ABB RobotStudio station: CeldaRobotica_PurpleWood.rsstnx

Station CeldaRobotica_PurpleWood (saved by RobotStudio 22.3.10190.2)
Controller Controlador1, task T_ROB1: task frame (RAPID world) sits at (-200, -100, 255) mm in the station
Controller Controlador1
  mechanical unit ROB_1: IRB1600_6_145__02, 6 joints, base frame (0, 0, 0) mm
Layout (positions relative to the parent item):
  - SC_Conveyor [smart component]
      signals: DI Crear_Gato, DI Crear_Estante, DI Crear_Mesa, DO DO_HIGH, DO DO_MID, DO DO_LOW, DO DO_GIRO
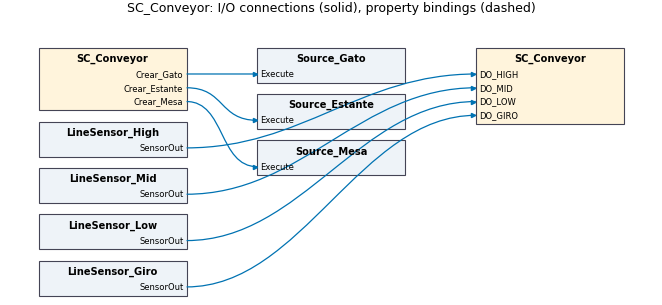
      connections:
        SC_Conveyor.Crear_Gato -> Source_Gato.Execute
        SC_Conveyor.Crear_Estante -> Source_Estante.Execute
        SC_Conveyor.Crear_Mesa -> Source_Mesa.Execute
        LineSensor_High.SensorOut -> SC_Conveyor.DO_HIGH
        LineSensor_Mid.SensorOut -> SC_Conveyor.DO_MID
        LineSensor_Low.SensorOut -> SC_Conveyor.DO_LOW
        LineSensor_Giro.SensorOut -> SC_Conveyor.DO_GIRO
    - EstanteColgado [graphiccomponentgroup] at (1130, -1000, 1506.1) mm, rotated rx 0 ry 0 rz 90 deg
      - RepisaLego:1 [graphiccomponentgroup] at (-95.35, -24.33, -484.95) mm, rotated rx 90 ry 86.54 rz -90 deg
        - RLV1 Fondo:1 [part] at (-151.16, -62.59, -80.25) mm, rotated rx 0 ry 90 rz 0 deg, size 66.4 x 11.1 x 483.7 mm
        - RLV1 Frente:1 [part] at (-151.16, -22.59, -49.25) mm, rotated rx 90 ry 0 rz 90 deg, size 83.3 x 30 x 483.3 mm
        - RLV1 Lateral:1 [part] at (-382.16, -18.58, -80.25) mm, rotated rx 180 ry 0 rz 180 deg, size 10.1 x 72.1 x 63.1 mm
        - RLV1 Trasera:1 [part] at (-151.16, -22.59, -111.25) mm, rotated rx -90 ry 0 rz 90 deg, size 91.4 x 15.2 x 487.6 mm
        - RLV1 Lateral:2 [part] at (88.84, -18.58, -80.25) mm, rotated rx 180 ry 0 rz 180 deg, size 10.1 x 72.1 x 63.1 mm
      - Gancho:1 [part] at (0, 0, -143.1) mm, size 142.1 x 142.1 x 242.6 mm
    - MesaColgada [graphiccomponentgroup] at (1130, -1000, 1506.1) mm, rotated rx 0 ry 0 rz 90 deg
      - AssemblyMesa2:1 [graphiccomponentgroup] at (0.6, -56.61, -255.15) mm, rotated rx -90 ry 79.48 rz -90 deg
        - MV1 Pata:1 [part] at (317.81, 42.68, -57.5) mm, size 36.5 x 51.1 x 116.8 mm
        - MV1 Tabla:1 [part] at (61.67, 51.7, 0) mm, rotated rx -90 ry 0 rz 0 deg, size 503.6 x 139.7 x 18.4 mm
        - MV1 Pata_MIR:1 [part] at (-194.43, 42.68, -57.5) mm, rotated rx 180 ry 0 rz 180 deg, size 36.5 x 51.1 x 116.8 mm
      - Gancho:1 [part] at (0, 0, -143.1) mm, size 142.1 x 142.1 x 242.6 mm
      - Source_Gato [smart component, from Components\Source.rslib] at (1000, 1130, -1506.1) mm, rotated rx 0 ry 0 rz -90 deg
          properties: Source=(none); Copy=(none); Parent=(none); Position=[0 0 0]; Orientation=[0 0 0]; Transient=false; PhysicsBehavior=-1
    - CasaGatoColgada_2 [graphiccomponentgroup] at (1130, -1000, 1506.1) mm, rotated rx 0 ry 0 rz 90 deg
      - Gancho:1 [part] at (0, 0, -143.1) mm, size 142.1 x 142.1 x 242.6 mm
      - CGV1 Pieza Base:1 [part] at (-126.11, -5.04, -68.58) mm, rotated rx -1.14 ry 0 rz 0 deg, size 304.2 x 16.3 x 706.2 mm
    - Source_Mesa [smart component, from Components\Source.rslib]
        properties: Source=MesaColgada; Copy=(none); Parent=(none); Position=[1.13 -2.9 1.5061]; Orientation=[0 0 1.5707963267949]; Transient=true; PhysicsBehavior=3
    - Source_Estante [smart component, from Components\Source.rslib]
        properties: Source=EstanteColgado; Copy=(none); Parent=(none); Position=[1.13 -2.9 1.5061]; Orientation=[0 0 1.5707963267949]; Transient=true; PhysicsBehavior=3
    - PhysicsControl [smart component, from Components\PhysicsControl.rslib]
        properties: Object=ConveyorAux; Behavior=1; SurfaceVelocity=0.05
    - LineSensor_Low [smart component, from Components\LineSensor.rslib]
        properties: Start=[1.2 -0.8 0.8]; End=[1.1 -0.8 0.8]; Radius=0; SensedPart=(none); SensedPoint=[0 0 0]
      - _sensorPart_ [part], size 100 x 0 x 0 mm
    - LineSensor_Mid [smart component, from Components\LineSensor.rslib]
        properties: Start=[1.15 -0.8 0.95]; End=[1.1 -0.8 0.95]; Radius=0; SensedPart=(none); SensedPoint=[0 0 0]
      - _sensorPart_ [part], size 50 x 0 x 0 mm
    - LineSensor_High [smart component, from Components\LineSensor.rslib]
        properties: Start=[1.3 -0.8 0.95]; End=[1.2 -0.8 0.95]; Radius=0; SensedPart=(none); SensedPoint=[0 0 0]
      - _sensorPart_ [part], size 100 x 0 x 0 mm
    - Source_Gato [smart component, from Components\Source.rslib]
        properties: Source=CasaGatoColgada_2; Copy=(none); Parent=(none); Position=[1.13 -2.9 1.5061]; Orientation=[0 0 1.5707963267949]; Transient=true; PhysicsBehavior=3
    - PhysicsControl_2 [smart component, from Components\PhysicsControl.rslib]
        properties: Object=ConveyorAux2; Behavior=1; SurfaceVelocity=0.05
    - ConveyorAux [part], size 30 x 6000 x 30 mm
    - ConveyorAux2 [part], size 30 x 6000 x 30 mm
    - LineSensor_Giro [smart component, from Components\LineSensor.rslib]
        properties: Start=[1.2 0 1.55]; End=[1.1 0 1.55]; Radius=0; SensedPart=(none); SensedPoint=[0 0 0]
      - _sensorPart_ [part], size 100 x 0 x 0 mm
  - Robotpedestal1400_H240 [part, from Equipment\Robot Pedestal 1400 H240.rslib] at (-330, -100, 0) mm
  - IRB1600_6_145__02 [mechanism, from Robots\IRB1600_6_145_G_02.rslib] at (-200, -100, 255) mm; joint values [0.1049, 0.2988, -0.3505, -0.1652, 0.584, 0.1908] (rad or m)
  - Conveyor [part], size 71 x 6000 x 68 mm
  - MyNewTool [mechanism] at (806.29, 0, 1409) mm, rotated rx -180 ry 60 rz -180 deg
      TCP MyNewTool at (0, 0, 200) mm
      links: Pieza_1
  - Fence_2500 [graphiccomponentgroup, from Equipment\Fence_2500.rslib] at (800, 1500, 0) mm, rotated rx 0 ry 0 rz 90 deg
    - Body 1 [part, from Equipment\Fence_2500.rslib]
    - Body 2 [part, from Equipment\Fence_2500.rslib]
  - Fence_2500_2 [graphiccomponentgroup, from Equipment\Fence_2500.rslib] at (1500, -1000, 0) mm
    - Body 1 [part, from Equipment\Fence_2500.rslib]
    - Body 2 [part, from Equipment\Fence_2500.rslib]
  - Fence_2500_3 [graphiccomponentgroup, from Equipment\Fence_2500.rslib] at (-1800, -1000, 0) mm
    - Body 1 [part, from Equipment\Fence_2500.rslib]
    - Body 2 [part, from Equipment\Fence_2500.rslib]
  - Gate [graphiccomponentgroup, from Equipment\Fence_Gate.rslib] at (-300, -1800, 0) mm, rotated rx 0 ry 0 rz 90 deg
    - Body 1 [part, from Equipment\Fence_Gate.rslib]
    - Body 2 [part, from Equipment\Fence_Gate.rslib]
    - Body 3 [part, from Equipment\Fence_Gate.rslib]
  - Fence_740 [graphiccomponentgroup, from Equipment\Fence_740.rslib] at (-1800, -1750, 0) mm
    - Body 1 [part, from Equipment\Fence_740.rslib]
    - Body 2 [part, from Equipment\Fence_740.rslib]
  - Fence_740_2 [graphiccomponentgroup, from Equipment\Fence_740.rslib] at (500, -1800, 0) mm, rotated rx 0 ry 0 rz 90 deg
    - Body 1 [part, from Equipment\Fence_740.rslib]
    - Body 2 [part, from Equipment\Fence_740.rslib]
  - Fence_740_3 [graphiccomponentgroup, from Equipment\Fence_740.rslib] at (1500, -1800, 0) mm
    - Body 1 [part, from Equipment\Fence_740.rslib]
    - Body 2 [part, from Equipment\Fence_740.rslib]
  - IRC5_Singel-Cabinet [part, from Equipment\IRC5_Singel-Cabinet.rslib] at (-2350, -1400, 100) mm, rotated rx 90 ry 0 rz -90 deg
Attachment: MyNewTool is attached to IRB1600_6_145__02 / Link6
Station signals: DO Estado_Pistola
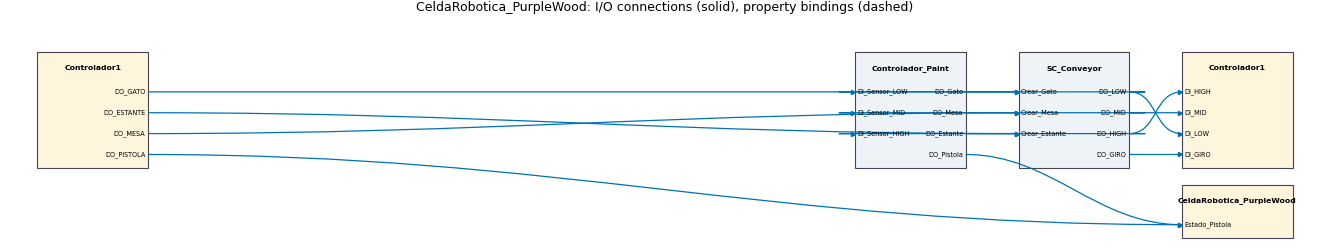
Station logic (signal -> signal, property => property):
  SC_Conveyor.DO_LOW -> Controlador_Paint.DI_Sensor_LOW
  SC_Conveyor.DO_MID -> Controlador_Paint.DI_Sensor_MID
  SC_Conveyor.DO_HIGH -> Controlador_Paint.DI_Sensor_HIGH
  Controlador_Paint.DO_Gato -> SC_Conveyor.Crear_Gato
  Controlador_Paint.DO_Mesa -> SC_Conveyor.Crear_Mesa
  Controlador_Paint.DO_Estante -> SC_Conveyor.Crear_Estante
  Controlador_Paint.DO_Pistola -> CeldaRobotica_PurpleWood.Estado_Pistola
  Controlador1.DO_GATO -> SC_Conveyor.Crear_Gato
  Controlador1.DO_ESTANTE -> SC_Conveyor.Crear_Estante
  Controlador1.DO_MESA -> SC_Conveyor.Crear_Mesa
  Controlador1.DO_PISTOLA -> CeldaRobotica_PurpleWood.Estado_Pistola
  SC_Conveyor.DO_HIGH -> Controlador1.DI_HIGH
  SC_Conveyor.DO_MID -> Controlador1.DI_MID
  SC_Conveyor.DO_LOW -> Controlador1.DI_LOW
  SC_Conveyor.DO_GIRO -> Controlador1.DI_GIRO
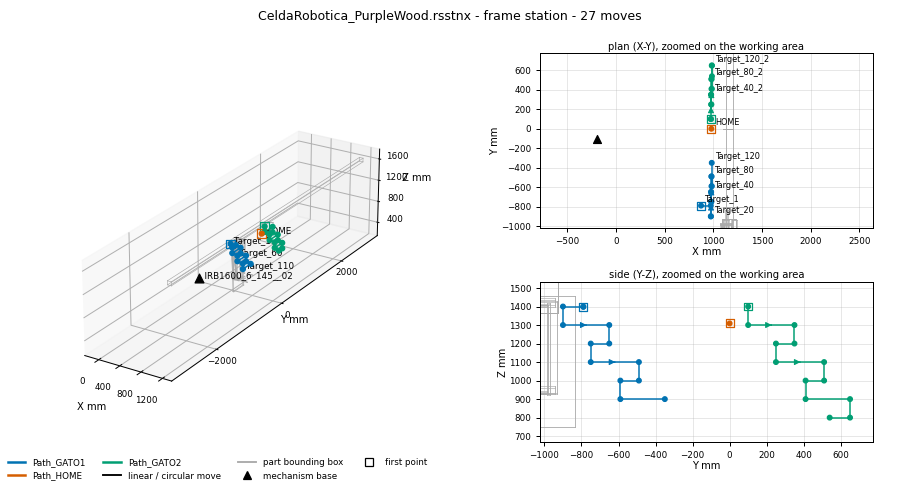
[picture p0: tool path of CeldaRobotica_PurpleWood.rsstnx in frame station, 27 of 27 moves have a stored position in this frame; points joined in program order, loops and branches not executed]
Targets, tools, work objects and paths stored in the station, written as RAPID:
! task T_ROB1
MODULE CalibData
  PERS tooldata TCP_TOOL:=[TRUE,[[0,0,200],[0.965925826,0,0.258819045,0]],[0.25,[0,0,1],[1,0,0,0],0,0,0]];
ENDMODULE

! task T_ROB1
MODULE CalibData
  PERS tooldata TCP_TOOL:=[TRUE,[[0,0,200],[0.965925826,0,0.258819045,0]],[0.25,[0,0,1],[1,0,0,0],0,0,0]];
ENDMODULE

! task T_ROB1
MODULE sysdata
  PERS tooldata tUserTool0:=[TRUE,[[0,0,0],[1,0,0,0]],[0.001,[0,0,0.001],[1,0,0,0],0,0,0]];
  PROC PowerOnWZones()
  ENDPROC
  PROC ConfSettingsOff()
    ConfJ \Off;
    ConfL \Off;
  ENDPROC
ENDMODULE

! task T_ROB1
MODULE robdata
  PERS tooldata tDefGun_Tip:=[TRUE,[[50,0,100],[0.866025,0,0.5,0]],[2,[0,0,50],[1,0,0,0],0,0,0]];
  PERS tooldata tDefGun_100:=[TRUE,[[136.6,0,150],[0.866025,0,0.5,0]],[2,[0,0,50],[1,0,0,0],0,0,0]];
  PERS tooldata tDefGun_200:=[TRUE,[[223.2,0,200],[0.866025,0,0.5,0]],[2,[0,0,50],[1,0,0,0],0,0,0]];
ENDMODULE

! task T_ROB1
MODULE pntexstart
  PROC ExStartReset()
  ENDPROC
  PROC WaitExStart()
    WaitTime 0.1;
  ENDPROC
ENDMODULE

! task T_ROB1
MODULE posmsg
  PROC PostMainPosMsg()
  ENDPROC
  PROC PreMainPosMsg()
  ENDPROC
ENDMODULE

! task T_ROB1
MODULE pntloop
  LOCAL VAR signaldo doJobCompAlias;
  PROC main()
    CallInitCustMain;
    ClearCurrentJob;
    Reset doJobCompAlias;
    PulseDO \High\PLength:=2.0,doJobCompAlias;
    ClearCurrentJob;
    WaitTime 0.2;
  ENDPROC
  LOCAL PROC ClearCurrentJob()
  ENDPROC
  PROC CallInitCustMain()
  ENDPROC
ENDMODULE

! task T_ROB1
MODULE custmain
  PROC PreMainCustom()
  ENDPROC
  PROC InitCustMain()
  ENDPROC
  PROC PostMainCustom()
  ENDPROC
ENDMODULE

! task T_ROB1
MODULE pntprogmap
  PROC SetProgramModule()
  ENDPROC
ENDMODULE

! task T_ROB1
MODULE pnttipclean
  PROC TipCleanPreMain()
    AppCleanRun;
    TipCleanRun;
    TipCleanRun;
    AppCleanRun;
  ENDPROC
  PROC TipCleanPostMain()
    AppCleanRun;
    TipCleanRun;
    TipCleanRun;
    AppCleanRun;
  ENDPROC
  PROC TipCleanRun()
  ENDPROC
  PROC AppCleanRun()
  ENDPROC
ENDMODULE

! task T_ROB1
MODULE CalibData
  TASK PERS wobjdata WO_GATO:=[FALSE,TRUE,"",[[1322.73,-1000,1198.166],[0.714094021,0,0.700049805,0]],[[0,0,0],[1,0,0,0]]];
  PERS tooldata TCP_TOOL:=[TRUE,[[0,0,200],[0.965925826,0,0.258819045,0]],[0.25,[0,0,1],[1,0,0,0],0,0,0]];
  PERS tooldata MyNewTool:=[TRUE,[[0,0,200],[1,0,0,0]],[1,[0,0,1],[1,0,0,0],0,0,0]];
  TASK PERS wobjdata WO_GATO_2:=[FALSE,TRUE,"",[[1322.73,0,1198.166],[0.714094021,0,0.700049805,0]],[[0,0,0],[1,0,0,0]]];
ENDMODULE

! task T_ROB1
MODULE Module1
  CONST robtarget HOME:=[[1179.496732003,100,1054],[0.258819045,0,0.965925826,0],[0,0,0,0],[9E+09,9E+09,9E+09,9E+09,9E+09,9E+09]];
  CONST robtarget Target_10:=[[50,310,-150],[1,0,0,0],[-1,1,-2,0],[9E+09,9E+09,9E+09,9E+09,9E+09,9E+09]];
  CONST robtarget Target_20:=[[50,200,-150],[1,0,0,0],[-1,1,-2,0],[9E+09,9E+09,9E+09,9E+09,9E+09,9E+09]];
  CONST robtarget Target_30:=[[150,200,-150],[1,0,0,0],[-1,1,-2,0],[9E+09,9E+09,9E+09,9E+09,9E+09,9E+09]];
  CONST robtarget Target_40:=[[150,450,-150],[1,0,0,0],[-1,1,-2,0],[9E+09,9E+09,9E+09,9E+09,9E+09,9E+09]];
  CONST robtarget Target_50:=[[250,450,-150],[1,0,0,0],[-1,1,-2,0],[9E+09,9E+09,9E+09,9E+09,9E+09,9E+09]];
  CONST robtarget Target_60:=[[250,350,-150],[1,0,0,0],[-1,1,-2,0],[9E+09,9E+09,9E+09,9E+09,9E+09,9E+09]];
  CONST robtarget Target_70:=[[350,350,-150],[1,0,0,0],[-1,1,-2,0],[9E+09,9E+09,9E+09,9E+09,9E+09,9E+09]];
  CONST robtarget Target_80:=[[350,610,-150],[1,0,0,0],[-1,1,-2,0],[9E+09,9E+09,9E+09,9E+09,9E+09,9E+09]];
  CONST robtarget Target_90:=[[450,610,-150],[1,0,0,0],[-1,1,-2,0],[9E+09,9E+09,9E+09,9E+09,9E+09,9E+09]];
  CONST robtarget Target_100:=[[450,510,-150],[1,0,0,0],[-1,1,-2,0],[9E+09,9E+09,9E+09,9E+09,9E+09,9E+09]];
  CONST robtarget Target_110:=[[550,510,-150],[1,0,0,0],[-1,1,-2,0],[9E+09,9E+09,9E+09,9E+09,9E+09,9E+09]];
  CONST robtarget Target_120:=[[550,750,-150],[1,0,0,0],[-1,1,-2,0],[9E+09,9E+09,9E+09,9E+09,9E+09,9E+09]];
  CONST robtarget Target_130:=[[650,750,-150],[1,0,0,0],[-1,1,-2,0],[9E+09,9E+09,9E+09,9E+09,9E+09,9E+09]];
  CONST robtarget Target_140:=[[650,640,-150],[1,0,0,0],[-1,1,-2,0],[9E+09,9E+09,9E+09,9E+09,9E+09,9E+09]];
  CONST robtarget Target_1:=[[50,310,-250],[1,0,0,0],[0,0,0,0],[9E+09,9E+09,9E+09,9E+09,9E+09,9E+09]];
  CONST robtarget Target_10_2:=[[50,310,-150],[1,0,0,0],[-1,1,-2,0],[9E+09,9E+09,9E+09,9E+09,9E+09,9E+09]];
  CONST robtarget Target_20_2:=[[50,200,-150],[1,0,0,0],[0,-2,1,0],[9E+09,9E+09,9E+09,9E+09,9E+09,9E+09]];
  CONST robtarget Target_30_2:=[[150,200,-150],[1,0,0,0],[0,-2,1,0],[9E+09,9E+09,9E+09,9E+09,9E+09,9E+09]];
  CONST robtarget Target_40_2:=[[150,450,-150],[1,0,0,0],[0,-2,1,0],[9E+09,9E+09,9E+09,9E+09,9E+09,9E+09]];
  CONST robtarget Target_50_2:=[[250,450,-150],[1,0,0,0],[0,-2,1,0],[9E+09,9E+09,9E+09,9E+09,9E+09,9E+09]];
  CONST robtarget Target_60_2:=[[250,350,-150],[1,0,0,0],[0,-2,1,0],[9E+09,9E+09,9E+09,9E+09,9E+09,9E+09]];
  CONST robtarget Target_70_2:=[[350,350,-150],[1,0,0,0],[0,-2,1,0],[9E+09,9E+09,9E+09,9E+09,9E+09,9E+09]];
  CONST robtarget Target_80_2:=[[350,610,-150],[1,0,0,0],[0,-2,1,0],[9E+09,9E+09,9E+09,9E+09,9E+09,9E+09]];
  CONST robtarget Target_90_2:=[[450,610,-150],[1,0,0,0],[0,-2,1,0],[9E+09,9E+09,9E+09,9E+09,9E+09,9E+09]];
  CONST robtarget Target_100_2:=[[450,510,-150],[1,0,0,0],[0,-2,1,0],[9E+09,9E+09,9E+09,9E+09,9E+09,9E+09]];
  CONST robtarget Target_110_2:=[[550,510,-150],[1,0,0,0],[0,-2,1,0],[9E+09,9E+09,9E+09,9E+09,9E+09,9E+09]];
  CONST robtarget Target_120_2:=[[550,750,-150],[1,0,0,0],[0,-2,1,0],[9E+09,9E+09,9E+09,9E+09,9E+09,9E+09]];
  CONST robtarget Target_130_2:=[[650,750,-150],[1,0,0,0],[0,-2,1,0],[9E+09,9E+09,9E+09,9E+09,9E+09,9E+09]];
  CONST robtarget Target_140_2:=[[650,640,-150],[1,0,0,0],[0,-2,1,0],[9E+09,9E+09,9E+09,9E+09,9E+09,9E+09]];
  PROC Path_GATO1()
    MoveJ Target_1,v1000,z100,MyNewTool\WObj:=WO_GATO;
    MoveL Target_10,v400,z100,MyNewTool\WObj:=WO_GATO;
    MoveL Target_20,v30,z100,MyNewTool\WObj:=WO_GATO;
    MoveL Target_30,v1000,z100,MyNewTool\WObj:=WO_GATO;
    MoveL Target_40,v800,z100,MyNewTool\WObj:=WO_GATO;
    MoveL Target_50,v1000,z100,MyNewTool\WObj:=WO_GATO;
    MoveL Target_60,v30,z100,MyNewTool\WObj:=WO_GATO;
    MoveL Target_70,v1000,z100,MyNewTool\WObj:=WO_GATO;
    MoveL Target_80,v800,z100,MyNewTool\WObj:=WO_GATO;
    MoveL Target_90,v1000,z100,MyNewTool\WObj:=WO_GATO;
    MoveL Target_100,v30,z100,MyNewTool\WObj:=WO_GATO;
    MoveL Target_110,v1000,z100,MyNewTool\WObj:=WO_GATO;
    MoveL Target_120,v800,z100,MyNewTool\WObj:=WO_GATO;
  ENDPROC
  PROC Path_HOME()
    MoveJ HOME,v1000,z100,TCP_TOOL\WObj:=wobj0;
  ENDPROC
  PROC main()
    Set DO_Gato;
    WaitTime 35;
    Reset DO_Gato;
    Set DO_Gato;
    Reset DO_Gato;
    Path_GATO1;
    Path_HOME;
    Path_GATO2;
    Path_HOME;
  ENDPROC
  PROC Path_GATO2()
    MoveL Target_20_2,v50,z100,MyNewTool\WObj:=WO_GATO_2;
    MoveL Target_30_2,v30,z100,MyNewTool\WObj:=WO_GATO_2;
    MoveL Target_40_2,v800,z100,MyNewTool\WObj:=WO_GATO_2;
    MoveL Target_50_2,v1000,z100,MyNewTool\WObj:=WO_GATO_2;
    MoveL Target_60_2,v30,z100,MyNewTool\WObj:=WO_GATO_2;
    MoveL Target_70_2,v1000,z100,MyNewTool\WObj:=WO_GATO_2;
    MoveL Target_80_2,v800,z100,MyNewTool\WObj:=WO_GATO_2;
    MoveL Target_90_2,v1000,z100,MyNewTool\WObj:=WO_GATO_2;
    MoveL Target_100_2,v30,z100,MyNewTool\WObj:=WO_GATO_2;
    MoveL Target_110_2,v1000,z100,MyNewTool\WObj:=WO_GATO_2;
    MoveL Target_120_2,v800,z100,MyNewTool\WObj:=WO_GATO_2;
    MoveL Target_130_2,v1000,z100,MyNewTool\WObj:=WO_GATO_2;
    MoveL Target_140_2,v30,z100,MyNewTool\WObj:=WO_GATO_2;
  ENDPROC
ENDMODULE

